(* IEC 61131-3 sources: horner-cscape-mcp/artifacts/projects/FailAudit_POU_LadderInjection/pous, 1 file *)

(* ---- POU_LadderInjection.st ---- *)
PROGRAM POU_LadderInjection
VAR
    StartSwitch : BOOL := TRUE;
END_VAR
---[ ]--- StartSwitch
END_PROGRAM
